{attribute 'qualified_only'}

TYPE incCommStates :
(
		stNull      :=    Consts.ST_NULL,
		stStartUp   :=    Consts.ST_START_UP,
		stInit      :=    Consts.ST_INIT,
		stReady     :=    Consts.ST_READY,
		stStop      :=    Consts.ST_STOP,
		stStepBlock :=    Consts.ST_STEP_BLOCK,	
		stEMG		:=    Consts.ST_EMG,
		
		
		stSetMode                := 1000,
		stStationStop,
		
		stIndexStart,
		stIndexEnableStations,
		stIndexStationsReady,
		stSignalStations,		
		stIndexEnable, 
		stIndexReady,
		stIndexCheck, 
		stIndexDone,
		
		stPurgeStart,
		stPurgeFinish,
		stPurgeDone,

		stErrCommFault

)DINT;
END_TYPE

(* stored: Version 1.1.0.1, ProductVersion 3.1.4024.3
   DUT incCommStates: Id {e605bfa2-28b8-491d-a5cc-4fd2d16c884a} *)
